Staubli VAL3: remEnableRem.pgx

program remEnableRem(string& sReturn[] (dimensions=1))
begin
  // Enable remote mode... remotely!
  //
  logMsg("call remEnableRem")
  bRemControlON=true
  sReturn="ENABLEREMOTE"
end
